FUNCTION_BLOCK AlarmCreatesVideo
VAR_INPUT
	ImageExportPath	: STRING(255);
	VideoFilePath	: STRING(255);
	JSONAttribute	: STRING;	
END_VAR
VAR_OUTPUT
	bBusy	: BOOL;
	bError	: BOOL;
	nErrID	: UDINT;
END_VAR
VAR
	Listener		: FB_ListenerBase2;
	JSONFilter		: FB_TcEventFilter;
	hr				: HRESULT;
	sJsonAttribute	: STRING;
	
	CreateVideo		: ImagesToVideo;
	CreateVideoFlag	: BOOL;
END_VAR

Listener.Execute();

//Filter out events using JSON attribute
JSONFilter.Clear().JsonAttribute.Value.EqualTo(JSONAttribute);
hr := Listener.Subscribe2(JSONFilter);

IF  sJsonAttribute = JSONAttribute THEN
	(*CreateVideo(
	bStart:= , 
	ImageExportPath:= , 
	VideoDestinationPath:= , 
	sFileName:= , 
	bBusy=> , 
	bError=> , 
	nErrID=> ); *)
	CreateVideoFlag := TRUE;
END_IF

END_FUNCTION_BLOCK

(* stored: Version 1.1.0.1, ProductVersion 3.1.4024.10
   POU AlarmCreatesVideo: Id {285e3901-0f5f-0d23-118c-3771e9af22f9}, SpecialFunc None *)
